(* CoDeSys 2.3.9.42 project: вижуал_тележки_94-95.pro *)
(* Libraries: Standard.lib 4.10.05 11:14:46, IecSfc.lib 13.4.06 15:51:28, SYSLIBCALLBACK.LIB 26.9.08 15:43:52 *)

(* Global variable list: Global_Variables *)
VAR_GLOBAL
	observer: BOOL;
	Warning: BOOL;
	Stop: BOOL;
	Start:BOOL;
END_VAR

(* POU PLC_PRG, FBD *)
PROGRAM PLC_PRG
VAR
	Trig1: R_TRIG;
	Trig2: F_TRIG;
	Timer1: TOF;
	Timer2: TON;
END_VAR
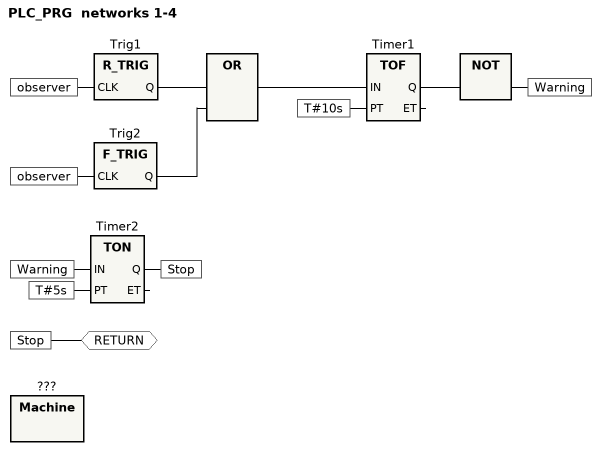
_FBD_ (* Function Block Diagram *)
NETWORK 1
	NOT Timer1:TOF(IN: OR(Trig1:R_TRIG(CLK: observer), Trig2:F_TRIG(CLK: observer)), PT: T#10s) => Warning
NETWORK 2
	Timer2:TON(IN: Warning, PT: T#5s) => Stop
NETWORK 3
	Stop => <RETURN>
NETWORK 4
	???:Machine()
_END_FBD_
END_PROGRAM

(* POU Machine, SFC *)
PROGRAM Machine
VAR
	X_pos: INT;
	Y_pos: INT;
	Counter: INT;
END_VAR
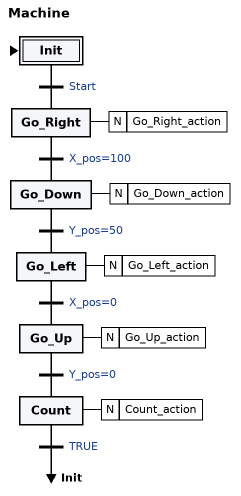
INITIAL_STEP Init:
END_STEP
TRANSITION FROM Init TO Go_Right := Start;
END_TRANSITION
STEP Go_Right:
	Go_Right_action(N);
END_STEP
TRANSITION FROM Go_Right TO Go_Down := X_pos=100;
END_TRANSITION
STEP Go_Down:
	Go_Down_action(N);
END_STEP
TRANSITION FROM Go_Down TO Go_Left := Y_pos=50;
END_TRANSITION
STEP Go_Left:
	Go_Left_action(N);
END_STEP
TRANSITION FROM Go_Left TO Go_Up := X_pos=0;
END_TRANSITION
STEP Go_Up:
	Go_Up_action(N);
END_STEP
TRANSITION FROM Go_Up TO Count := Y_pos=0;
END_TRANSITION
STEP Count:
	Count_action(N);
END_STEP
TRANSITION FROM Count TO Init := TRUE;
END_TRANSITION

ACTION Go_Right_action:
X_pos:=X_pos+1;
END_ACTION

ACTION Go_Down_action:
Y_pos:=Y_pos+1;
END_ACTION

ACTION Go_Left_action:
X_pos:=X_pos-1;
END_ACTION

ACTION Go_Up_action:
Y_pos:=Y_pos-1;
END_ACTION

ACTION Count_action:
Counter:=Counter+1;
END_ACTION
END_PROGRAM

(* Visualisation observation
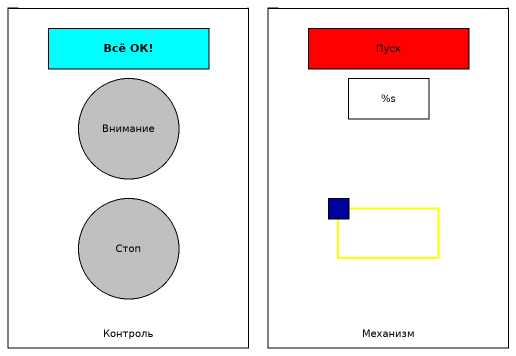
rectangle at (90,70)-(251,111): text "Всё ОК!"; alarm colour if .observer; taps .observer
rectangle at (350,70)-(511,111): text "Пуск"; alarm colour if .Start; taps .Start
ellipse at (120,120)-(221,221): text "Внимание"; alarm colour if .Warning
ellipse at (120,240)-(221,341): text "Стоп"; alarm colour if .Stop
rectangle at (390,120)-(471,161): text "%s"; shows Machine.Counter
rectangle at (90,360)-(251,391): text "Контроль"
rectangle at (350,360)-(511,391): text "Механизм"
rectangle at (370,240)-(391,261): x offset Machine.X_pos; y offset Machine.Y_pos
4 more shapes without text or variables
*)
